Staubli VAL3: setSizeList.pgx

public program setSizeList(num nPx (dimensions=1), num nPy (dimensions=1), num nPBottomX (dimensions=1), num nPBottomY (dimensions=1))
begin
  nTopX=nTopX[1]=nPx
  nTopY=nPy
  nBottomX=nBottomX[1]=nPBottomX
  nBottomY=nPBottomY
end
